FUNCTION_BLOCK FB_AxisSetSlaveState
VAR_INPUT
	bExecute: BOOL;
	stHardware: ST_AxisHardware;
	reqState: WORD;
END_VAR
VAR_OUTPUT
	bDone: BOOL;
	bBusy: BOOL;
	bError: BOOL;
	nErrId: UDINT;
	currStateDrive: ST_EcSlaveState;
	currStateEnc: ST_EcSlaveState;
END_VAR
VAR
	fbDriveState: FB_EcSetSlaveState;
	fbEncState: FB_EcSetSlaveState;
	bBusyDrive: BOOL;
	bBusyEnc: BOOL;
	bErrorDrive: BOOL;
	bErrorEnc: BOOL;
	nErrIdDrive: UDINT;
	nErrIdEnc: UDINT;
END_VAR

// Transition terminals if they exist
IF stHardware.drive_type > 0 THEN
	fbDriveState(sNetID:=stHardware.drive_ref.sNetId,
		nSlaveAddr:=stHardware.drive_ref.nSlaveAddr,
		bExecute:=bExecute,
		reqState:=reqState,
		bBusy=>bBusyDrive,
		bError=>bErrorDrive,
		nErrId=>nErrIdDrive,
		currState=>currStateDrive);
ELSE
	bBusyDrive := FALSE;
	bErrorDrive := FALSE;
	nErrIdDrive := 0;
END_IF
IF stHardware.enc_type > 0 THEN
	fbEncState(sNetID:=stHardware.enc_ref.sNetId,
		nSlaveAddr:=stHardware.enc_ref.nSlaveAddr,
		bExecute:=bExecute,
		reqState:=reqState,
		bBusy=>bBusyDrive,
		bError=>bErrorDrive,
		nErrId=>nErrIdDrive,
		currState=>currStateEnc);
ELSE
	bBusyEnc := FALSE;
	bErrorEnc := FALSE;
	nErrIdDrive := 0;
END_IF
bBusy := bBusyDrive OR bBusyEnc;
bDone := bExecute AND NOT bBusy;
bError := bErrorDrive OR bErrorEnc;
IF nErrIdDrive > 0 THEN
	nErrId := nErrIdDrive;
ELSE
	nErrId := nErrIdEnc;
END_IF

END_FUNCTION_BLOCK

(* stored: Version 1.1.0.1, ProductVersion 3.1.4020.14
   POU FB_AxisSetSlaveState: Id {826b3849-ce16-4717-9daa-1c853595336a}, SpecialFunc None *)
